Yaskawa INFORM job: USER_CART_S1.JBI

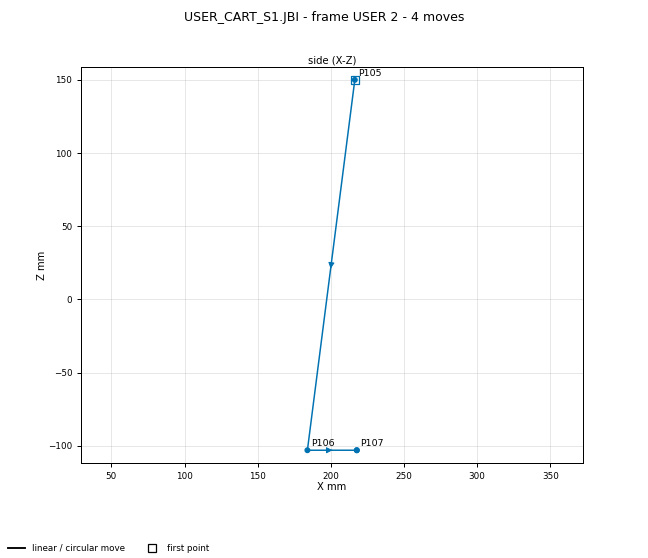
[picture p0: tool path of USER_CART_S1.JBI in frame USER 2, 4 of 4 moves have a stored position in this frame; points joined in program order, loops and branches not executed]
/JOB
//NAME USER_CART_S1
//POS
///NPOS 0,0,0,4,0,0
///TOOL 0
///USER 2
///POSTYPE USER
///RECTAN
///RCONF 1,0,0,0,0,0,0,0,0,0,0,0,0,0,0,0,0,0,0,0,0,0,0,0
P00105=216.374,-55.365,150.000,179.9941,-0.0013,-179.9943
P00106=183.974,-55.386,-103.111,179.9969,-0.0014,-179.9945
P00107=217.725,-55.392,-103.109,179.9979,-0.0019,-179.9959
P00108=217.733,-59.426,-103.121,179.9979,-0.0009,-179.9957
//INST
///DATE 2026/08/22 00:00
///ATTR SC,RW
///GROUP1 RB1
NOP
MOVJ P105 VJ=25.00
MOVL P106 V=150.0
MOVL P107 V=150.0
MOVL P108 V=150.0
END
